// TIA Portal V17 export
// export: Created 2024-09-03T21:54:47.4568105Z, ExportSetting WithDefaults, DisplayName Totally Integrated Automation Portal, DisplayVersion V17 Update 7, DisplayName TIA Portal Openness, DisplayVersion V17 Update 7, DisplayName TIA Portal Version Control Interface, DisplayVersion V17, DisplayName SINAMICS Startdrive Advanced, DisplayVersion V17 SP2, DisplayName SINAMICS Startdrive G110M, G120, G120C, G120D, G120P, G115D, DisplayVersion V17 SP2, DisplayName SINAMICS Startdrive G130, G150, S120, S150, SINAMICS MV, S210, DisplayVersion V17 SP2, DisplayName STEP 7 Professional, DisplayVersion V17 Update 7, DisplayName STEP 7 Safety, DisplayVersion V17 Update 6, DisplayName WinCC Advanced / Unified PC, DisplayVersion V17 Update 7
DATA_BLOCK "SlidesMain_DB"   // DB45
VERSION : 0.1
// stored: AutoNumber true, DBAccessibleFromOPCUA true, DBAccessibleFromWebserver true, InstanceOfName SlidesMain, InstanceOfType FB
"SlidesMain"
   // VAR
   //    R_TRIG_Instance { S7_SetPoint := 'True'} : R_TRIG;
   //    IEC_Timer_0_Instance { S7_SetPoint := 'True'} : TON_TIME;
   //    IEC_Timer_0_Instance_1 { S7_SetPoint := 'True'} : TOF_TIME;
   //    IEC_Timer_0_Instance_3 { S7_SetPoint := 'True'} : TON_TIME;
   //    IEC_Timer_0_Instance_5 { S7_SetPoint := 'True'} : TON_TIME;
   // END_VAR
BEGIN
   R_TRIG_Instance.CLK := FALSE;
   R_TRIG_Instance.Q := FALSE;
   R_TRIG_Instance.Stat_Bit := FALSE;
   IEC_Timer_0_Instance.PT := T#0MS;
   IEC_Timer_0_Instance.IN := FALSE;
   IEC_Timer_0_Instance_1.PT := T#0MS;
   IEC_Timer_0_Instance_1.IN := TRUE;
   IEC_Timer_0_Instance_3.PT := T#0MS;
   IEC_Timer_0_Instance_3.IN := FALSE;
   IEC_Timer_0_Instance_5.PT := T#0MS;
   IEC_Timer_0_Instance_5.IN := FALSE;
END_DATA_BLOCK
